FUNCTION_BLOCK FB_ServoMotor IMPLEMENTS I_ServoMotor
VAR_INPUT
END_VAR
VAR_OUTPUT
END_VAR
VAR
END_VAR

{warning 'Add method implementation '}
METHOD BeweegNaarDoel
VAR_INPUT
	IDoelPositie	: INT;
END_VAR

VAR
	IPositie : INT;
	TONBeweegTimer : TON := (PT:= T#1S, IN:= TONVariabele);
	TONVariabele : BOOL;
END_VAR

VAR CONSTANT
	IMotorSnelheid : INT := 5; 
END_VAR
IF TONBeweegTimer.Q = 1 AND MotorStatus = 1 THEN
	IF IDoelPositie > IPositie THEN
		IPositie:= IPositie + IMotorSnelheid;
	ELSIF IDoelPositie < IPositie THEN
		IPositie:= IPositie - IMotorSnelheid;
	ELSIF IDoelPositie = IPositie THEN // code fix voor overshoot
		IPositie:= IDoelPositie;
		
	END_IF
	
	TONVariabele := 1;
	
ELSIF TONBeweegTimer.Q = 0 AND TONVariabele =  1 AND MotorStatus = 1 THEN
	TONVariabele := 0;
END_IF
END_METHOD

PROPERTY MotorStatus : E_MotorStatus
GET
END_GET
SET
END_SET
END_PROPERTY

{warning 'Add property implementation'}
PROPERTY Positie : INT
GET
END_GET
END_PROPERTY

{warning 'Add method implementation '}
METHOD Start
END_METHOD

{warning 'Add method implementation '}
METHOD Stop
END_METHOD

END_FUNCTION_BLOCK

(* stored: Version 1.1.0.1
   POU FB_ServoMotor: Id {63955412-bcd3-4783-ab58-d217a713d49f}, SpecialFunc None
   Method BeweegNaarDoel: Id {3aa19c92-d64d-4fa9-b144-f711e11a9595}
   Property MotorStatus: Id {f3515037-d7f1-4cdf-986c-5e4909665074}
   Get Get: Id {27bff63a-6d8b-446e-b4a2-550c7791f64a}
   Set Set: Id {b4817821-45b4-4de7-bd99-86450dd53a84}
   Property Positie: Id {3f190714-8df9-4d2a-abfe-e5a5df771a72}
   Get Get: Id {2efa94e1-195f-4ab4-81b1-0730edbf470f}
   Method Start: Id {364a46ee-36a0-4191-aedb-115fa39384d7}
   Method Stop: Id {846d696b-ac2e-4b42-90ea-009facad47ec} *)
